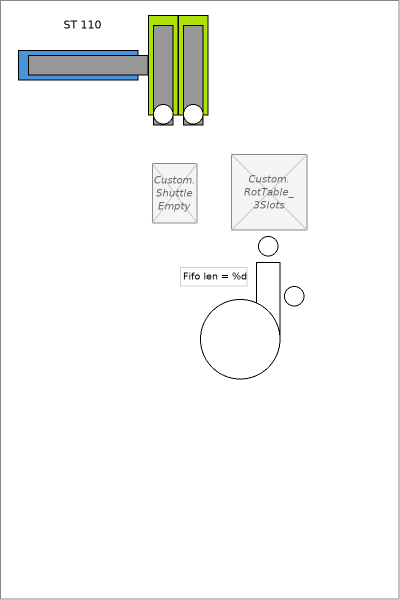
VISUALIZATION VISU_ST110  // 400x600
    Image (152,163 45x60), invisible if: NOT __ISVALIDREF(GVL._Process2._Mover), image: Custom.Shuttle Empty
    Image (231,154 76x76), image: Custom.RotTable_3Slots
        p2858320360: ST110_Axis.axis110_10W.axis.NcToPlc.ModuloActPos
    Rectangle (18,50 120x30)
    Rectangle (28,55 120x20)
        p3560616238: GVL._Process2.fb_Pnp.fb_simu_axis110_01Y.rOUT_PixActual
    Rectangle (148,15 30x100)
        p3560616238: GVL._Process2.fb_Pnp.fb_simu_axis110_01Y.rOUT_PixActual
    Rectangle (153,25 20x100)
        p2738717112: GVL._Process2.fb_Pnp.fb_simu_axis110_02Z.rOUT_PixActual
        p3560616238: GVL._Process2.fb_Pnp.fb_simu_axis110_01Y.rOUT_PixActual
    Rectangle (178,15 30x100)
        p3560616238: GVL._Process2.fb_Pnp.fb_simu_axis110_01Y.rOUT_PixActual
    Rectangle (183,25 20x100)
        p2738717112: GVL._Process2.fb_Pnp.fb_simu_axis110_03Z.rOUT_PixActual
        p3560616238: GVL._Process2.fb_Pnp.fb_simu_axis110_01Y.rOUT_PixActual
    Rectangle (256,262 24x73)
    Ellipse (200,299 80x80), colour toggle: GVL._Process2.fb_Feeder.simu_feeder.xIN_Enable
    Ellipse (284,286 20x20), colour toggle: GVL._Process2.fb_Feeder.simu_feeder.xOUT_NewPiece
    Ellipse (153,104 20x20)
        p3560616238: GVL._Process2.fb_Pnp.fb_simu_axis110_01Y.rOUT_PixActual
        p2738717112: GVL._Process2.fb_Pnp.fb_simu_axis110_02Z.rOUT_PixActual
    Ellipse (183,104 20x20)
        p2738717112: GVL._Process2.fb_Pnp.fb_simu_axis110_02Z.rOUT_PixActual
        p3560616238: GVL._Process2.fb_Pnp.fb_simu_axis110_01Y.rOUT_PixActual
    Ellipse (258,236 20x20), colour toggle: NOT GVL._Process2.fb_Feeder.simu_fifo.IsEmpty()
    Textfield (180,267 67x19), "Fifo len = %d", text variable: GVL._Process2.fb_Feeder.simu_fifo.GetLen()
    Label (40,15 85x20), "ST 110"
END_VISUALIZATION

(* stored: Version 1.1.0.1, ProductVersion 3.1.4024.6
   Visu VISU_ST110: Id {e87517ac-fb2f-4d50-b21f-e5c3a310ec53} *)
